// TIA Portal V17 export
// export: Created 2022-07-20T06:59:44.9663361Z, ExportSetting WithDefaults, DisplayName Totally Integrated Automation Portal, DisplayVersion V17, DisplayName TIA Portal Openness, DisplayVersion V17, DisplayName TIA Portal Version Control Interface, DisplayVersion V17, DisplayName SINAMICS Startdrive Advanced, DisplayVersion V17, DisplayName SINAMICS Startdrive G130, G150, S120, S150, SINAMICS MV, S210, DisplayVersion V17, DisplayName SINAMICS Startdrive G110M, G120, G120C, G120D, G120P, G115D, DisplayVersion V17, DisplayName STEP 7 Professional, DisplayVersion V17, DisplayName STEP 7 Safety, DisplayVersion V17, DisplayName WinCC Advanced, DisplayVersion V17
FUNCTION_BLOCK "FB10079_UvDryer"   // FB10079, LAD
{ S7_Optimized_Access := 'TRUE' }
VERSION : 0.1
// stored: AutoNumber false, IsIECCheckEnabled false, IsRetainMemResEnabled false, MemoryReserve 100, SetENOAutomatically false, UDAEnableTagReadback false
   VAR_INPUT
      UvDryer_Disable : Bool;
      Shutter_MotorInError : Bool;
      Shutter_PWMSetPoint : Real;
      Shutter_SensorClosed : Bool;
      Shutter_RequestInitialization : Bool;
      Shutter_RequestOpen : Bool;
      Shutter_RequestClose : Bool;
      Shutter_PWMCardInError : Bool;
      AirExtractor_ScalingShutterOpen : "stAirExtractorScalingParameters";
      AirExtractor_ScalingShutterClosed : "stAirExtractorScalingParameters";
      AirExtractor_PWMMinFrequenceValue : Real;
      AirExtractor_PWMMaxFrequenceValue : Real;
      AirExtractor_RequestActive : Bool;
      UvLamp_ThermalFuse : Bool;
      UvLamp_LampReady : Bool;
      UvLamp_LampWarning : Bool;
      UvLamp_LampError : Bool;
      UvLamp_FeedbackTensionOrErrorCode : Int;
      UvLamp_SetPoint : Real;
      TransportActivated : Bool;
      PowerOnBay : Bool;
   END_VAR
   VAR_OUTPUT
      Shutter_InitializeShutter : Bool;
      Shutter_OpenShutter : Bool;
      Shutter_CloseShutter : Bool;
      Shutter_PWMValue : Real;
      Shutter_ResetPWMCard : Bool;
      Shutter_InError : Bool;
      Shutter_Initialized : Bool;
      Shutter_Opened : Bool;
      Shutter_Closed : Bool;
      AirExtractor_Active : Bool;
      AirExtractor_PWMValue : Real;
      AirExtractor_AnalogValue : Int;
      UvLamp_ActiveLamp : Bool;
      UvLamp_ActivePowerRelay : Bool;
      UvLamp_AnalogValue : Int;
      UvLamp_WarmingUp : Bool;
      UvLamp_ErrorCode : Int;
      UvDryer_Disabled : Bool;
      UvDryer_Ready : Bool;
      UvDryer_Warning : Bool;
      UvDryer_Error : Bool;
      UvDryer_ShutdownInProgress : Bool;
      UvDryer_ShutdownDone : Bool;
      UvDryer_ShutdownTime : Time;
   END_VAR
   VAR_IN_OUT
      UvDryer_RequestStartDryer : Bool;
      UvDryer_RequestShutdown : Bool;
   END_VAR
   VAR
      ShutterMovementManagementStateDiagram : Int;
      DisableShutterStateDiagram : Int;
      AirExtractorManagementStateDiagram : Int;
      R_TRIG_UvDryerDisable : R_TRIG;
      R_TRIG_RequestStartDryer : R_TRIG;
      R_TRIG_ShutterSensorClosed { S7_SetPoint := 'True'} : R_TRIG;
      R_TRIG_RequestInitializeShutter { S7_SetPoint := 'True'} : R_TRIG;
      R_TRIG_RequestOpenShutter { S7_SetPoint := 'True'} : R_TRIG;
      R_TRIG_RequestCloseShutter { S7_SetPoint := 'True'} : R_TRIG;
      R_TRIG_RequestActiveAirExtractor { S7_SetPoint := 'True'} : R_TRIG;
      R_TRIG_RequestShutDown { S7_SetPoint := 'True'} : R_TRIG;
      F_TRIG_RequestStartDryer : F_TRIG;
      F_TRIG_RequestActiveAirExtractor { S7_SetPoint := 'True'} : F_TRIG;
      F_TRIG_PowerOnBay { S7_SetPoint := 'True'} : F_TRIG;
      F_TRIG_TransportActivated { S7_SetPoint := 'True'} : F_TRIG;
      F_TRIG_ShutterSensorClose { S7_SetPoint := 'True'} : F_TRIG;
      F_TRIG_ShutterMotorInError { S7_SetPoint := 'True'} : F_TRIG;
      F_TRIG_UvDryerInError { S7_SetPoint := 'True'} : F_TRIG;
      TON_ShutdownTimer { S7_SetPoint := 'True'} : TON_TIME;
      TON_ShutterMovement { S7_SetPoint := 'True'} : TON_TIME;
      FB10073_LampUVErrorManager_Instance { S7_SetPoint := 'True'} : "FB10073_LampUVErrorManager";
      UvLamp_FeedbackTensionVolts : Real;
      UvLamp_FeedbackTensionPrctg : Real;
   END_VAR
   VAR CONSTANT
      WAIT_FOR_MOVEMENT_REQUEST : Int := 0;
      INITIALIZE_SHUTTER : Int := 10;
      OPEN_SHUTTER : Int := 20;
      CLOSE_SHUTTER : Int := 30;
      MOVEMENT_DONE : Int := 40;
      "==========" : Bool;
      WAIT_FOR_AIR_EXTRACTOR_REQUEST : Int := 0;
      ACTIVE_AIR_EXTRACTOR : Int := 10;
      SHUTDOWN_AIR_EXTRACTOR_IN_PROGRESS : Int := 20;
      ACTIVE_MANUAL_AIR_EXTRACTOR : Int := 30;
      REQUEST_DONE : Int := 40;
   END_VAR
BEGIN

REGION Network 1 (SCL): First Scan
   IF "FirstScan" THEN
       #Shutter_Initialized := FALSE;
       #Shutter_Opened := FALSE;
       #Shutter_Closed := FALSE;
       #ShutterMovementManagementStateDiagram := 0;
   END_IF;
END_REGION

REGION Network 2 (SCL): Edge Signals & Timers
   REGION EDGE SIGNALS
       #R_TRIG_UvDryerDisable(CLK := #UvDryer_Disable);
       #R_TRIG_RequestStartDryer(CLK := #UvDryer_RequestStartDryer AND NOT(#UvDryer_ShutdownInProgress));
       #R_TRIG_RequestInitializeShutter(CLK := #Shutter_RequestInitialization);
       #R_TRIG_RequestOpenShutter(CLK := #Shutter_RequestOpen);
       #R_TRIG_RequestCloseShutter(CLK := #Shutter_RequestClose);
       #R_TRIG_ShutterSensorClosed(CLK := #Shutter_SensorClosed);
       #R_TRIG_RequestShutDown(CLK := #UvDryer_RequestShutdown);
       #R_TRIG_RequestActiveAirExtractor(CLK := #AirExtractor_RequestActive);

       #F_TRIG_RequestStartDryer(CLK := #UvDryer_RequestStartDryer);
       #F_TRIG_RequestActiveAirExtractor(CLK := #AirExtractor_RequestActive);
       #F_TRIG_PowerOnBay(CLK := #PowerOnBay);
       #F_TRIG_TransportActivated(CLK := #TransportActivated);
       #F_TRIG_ShutterSensorClose(CLK := #Shutter_SensorClosed);
       #F_TRIG_UvDryerInError(CLK := #UvDryer_Error);
       #F_TRIG_ShutterMotorInError(CLK := #Shutter_InError);
   END_REGION

   REGION TIMERS
       #TON_ShutdownTimer(IN := #UvDryer_ShutdownInProgress AND #PowerOnBay,
                          PT := T#5m,
                          ET => #UvDryer_ShutdownTime);
       #TON_ShutterMovement(IN := (#ShutterMovementManagementStateDiagram = #INITIALIZE_SHUTTER) OR
                            (#ShutterMovementManagementStateDiagram = #OPEN_SHUTTER) OR
                            (#ShutterMovementManagementStateDiagram = #CLOSE_SHUTTER),
                            PT := T#10s);
   END_REGION
END_REGION

REGION Network 3 (SCL): Uv Dryer Commands Management
   IF #F_TRIG_PowerOnBay.Q OR #F_TRIG_UvDryerInError.Q OR #F_TRIG_ShutterMotorInError.Q OR #UvDryer_Disable OR #UvDryer_ShutdownInProgress THEN
       #UvDryer_RequestStartDryer := FALSE;
   END_IF;
END_REGION

REGION Network 4 (SCL): Shutter Management
   CASE #ShutterMovementManagementStateDiagram OF
       #WAIT_FOR_MOVEMENT_REQUEST:
           IF (#R_TRIG_RequestStartDryer.Q OR #R_TRIG_RequestInitializeShutter.Q) AND NOT (#UvDryer_Disable) THEN
               #ShutterMovementManagementStateDiagram := #INITIALIZE_SHUTTER;
           ELSIF #R_TRIG_RequestOpenShutter.Q AND #Shutter_SensorClosed AND #TransportActivated AND #Shutter_Initialized THEN
               #Shutter_Opened := FALSE;
               #Shutter_Closed := FALSE;
               #ShutterMovementManagementStateDiagram := #OPEN_SHUTTER;
           ELSIF (#R_TRIG_RequestCloseShutter.Q OR #F_TRIG_TransportActivated.Q OR (#R_TRIG_UvDryerDisable.Q AND #Shutter_InError)) AND NOT (#Shutter_SensorClosed) THEN
               #Shutter_Opened := FALSE;
               #Shutter_Closed := FALSE;
               #ShutterMovementManagementStateDiagram := #CLOSE_SHUTTER;
           END_IF;
       #INITIALIZE_SHUTTER:
           #Shutter_InitializeShutter := TRUE;
           #Shutter_PWMValue := #Shutter_PWMSetPoint;
           IF #R_TRIG_ShutterSensorClosed.Q THEN
               RESET_TIMER(#TON_ShutterMovement);
               #Shutter_InitializeShutter := FALSE;
               #Shutter_Initialized := TRUE;
               #Shutter_Opened := FALSE;
               #Shutter_Closed := TRUE;
               #ShutterMovementManagementStateDiagram := #MOVEMENT_DONE;
           END_IF;
       #OPEN_SHUTTER:
           #Shutter_OpenShutter := TRUE;
           #Shutter_PWMValue := #Shutter_PWMSetPoint;
           IF #F_TRIG_ShutterSensorClose.Q THEN
               RESET_TIMER(#TON_ShutterMovement);
               #Shutter_OpenShutter := FALSE;
               #Shutter_Opened := TRUE;
               #Shutter_Closed := FALSE;
               #ShutterMovementManagementStateDiagram := #MOVEMENT_DONE;
           END_IF;
       #CLOSE_SHUTTER:
           #Shutter_CloseShutter := TRUE;
           #Shutter_PWMValue := #Shutter_PWMSetPoint;
           IF #R_TRIG_ShutterSensorClosed.Q THEN
               RESET_TIMER(#TON_ShutterMovement);
               #Shutter_CloseShutter := FALSE;
               #Shutter_Opened := FALSE;
               #Shutter_Closed := TRUE;
               #ShutterMovementManagementStateDiagram := #MOVEMENT_DONE;
           END_IF;
       #MOVEMENT_DONE:
           #ShutterMovementManagementStateDiagram := #WAIT_FOR_MOVEMENT_REQUEST;
   END_CASE;
END_REGION

REGION Network 5 (SCL): Air Extractor Management
   IF #R_TRIG_RequestStartDryer.Q AND NOT (#UvDryer_Disable) THEN
       #UvDryer_ShutdownDone := FALSE;
       #AirExtractorManagementStateDiagram := #ACTIVE_AIR_EXTRACTOR;
   ELSIF
       (#R_TRIG_RequestShutDown.Q AND NOT (#UvDryer_Disabled)) OR
       (#F_TRIG_RequestStartDryer.Q AND NOT (#UvDryer_Disabled)) OR
       (#R_TRIG_UvDryerDisable.Q AND (#AirExtractorManagementStateDiagram = #ACTIVE_AIR_EXTRACTOR OR #AirExtractorManagementStateDiagram = #ACTIVE_MANUAL_AIR_EXTRACTOR))
   THEN
       #AirExtractorManagementStateDiagram := #SHUTDOWN_AIR_EXTRACTOR_IN_PROGRESS;
   END_IF;

   CASE #AirExtractorManagementStateDiagram OF
       #WAIT_FOR_AIR_EXTRACTOR_REQUEST:
           #UvDryer_ShutdownInProgress := FALSE;
           #AirExtractor_Active := FALSE;
           #AirExtractor_PWMValue := 0;
           #AirExtractor_AnalogValue := 0;

           IF #R_TRIG_RequestActiveAirExtractor.Q AND NOT(#UvDryer_Disable) THEN
               #UvDryer_ShutdownDone := FALSE;
               #AirExtractorManagementStateDiagram := #ACTIVE_MANUAL_AIR_EXTRACTOR;
           END_IF;
       #ACTIVE_AIR_EXTRACTOR:
           #AirExtractor_Active := TRUE;
           IF #Shutter_Closed THEN
               "FC10072_ScalingAirExtraction_VolatgeFeedback"(VoltageFeedback := #UvLamp_FeedbackTensionVolts,
                                                              X_UVPower_Min := #AirExtractor_ScalingShutterClosed.PowerXMin,
                                                              X_UVPower_Max := #AirExtractor_ScalingShutterClosed.PowerXMax,
                                                              Y_AirPower_Min := #AirExtractor_ScalingShutterClosed.PowerAirYMin,
                                                              Y_AirPower_Max := #AirExtractor_ScalingShutterClosed.PowerAirYMax,
                                                              PWM_Minimum := #AirExtractor_PWMMinFrequenceValue,
                                                              PWM_Maximum := #AirExtractor_PWMMaxFrequenceValue,
                                                              Analogical_Value => #AirExtractor_AnalogValue,
                                                              PWM_FrequenceValue => #AirExtractor_PWMValue);
           ELSIF #Shutter_Opened THEN
               "FC10072_ScalingAirExtraction_VolatgeFeedback"(VoltageFeedback := #UvLamp_FeedbackTensionVolts,
                                                              X_UVPower_Min := #AirExtractor_ScalingShutterOpen.PowerXMin,
                                                              X_UVPower_Max := #AirExtractor_ScalingShutterOpen.PowerXMax,
                                                              Y_AirPower_Min := #AirExtractor_ScalingShutterOpen.PowerAirYMin,
                                                              Y_AirPower_Max := #AirExtractor_ScalingShutterOpen.PowerAirYMax,
                                                              PWM_Minimum := #AirExtractor_PWMMinFrequenceValue,
                                                              PWM_Maximum := #AirExtractor_PWMMaxFrequenceValue,
                                                              Analogical_Value => #AirExtractor_AnalogValue,
                                                              PWM_FrequenceValue => #AirExtractor_PWMValue);
           END_IF;


           IF #R_TRIG_RequestShutDown.Q OR #F_TRIG_RequestStartDryer.Q THEN
               #AirExtractorManagementStateDiagram := #SHUTDOWN_AIR_EXTRACTOR_IN_PROGRESS;
           END_IF;
       #SHUTDOWN_AIR_EXTRACTOR_IN_PROGRESS:
           #AirExtractor_Active := TRUE;

           "FC10072_ScalingAirExtraction_VolatgeFeedback"(VoltageFeedback := #AirExtractor_ScalingShutterClosed.PowerXMax,
                                                          X_UVPower_Min := #AirExtractor_ScalingShutterClosed.PowerXMin,
                                                          X_UVPower_Max := #AirExtractor_ScalingShutterClosed.PowerXMax,
                                                          Y_AirPower_Min := #AirExtractor_ScalingShutterClosed.PowerAirYMin,
                                                          Y_AirPower_Max := #AirExtractor_ScalingShutterClosed.PowerAirYMax,
                                                          PWM_Minimum := #AirExtractor_PWMMinFrequenceValue,
                                                          PWM_Maximum := #AirExtractor_PWMMaxFrequenceValue,
                                                          Analogical_Value => #AirExtractor_AnalogValue,
                                                          PWM_FrequenceValue => #AirExtractor_PWMValue);
           IF #TON_ShutdownTimer.Q THEN
               #AirExtractor_Active := FALSE;
               #UvDryer_ShutdownDone := TRUE;
               #AirExtractorManagementStateDiagram := #REQUEST_DONE;
           END_IF;
       #ACTIVE_MANUAL_AIR_EXTRACTOR:
           #AirExtractor_Active := TRUE;
           "FC10072_ScalingAirExtraction_VolatgeFeedback"(VoltageFeedback := #AirExtractor_ScalingShutterClosed.PowerXMin,
                                                          X_UVPower_Min := #AirExtractor_ScalingShutterClosed.PowerXMin,
                                                          X_UVPower_Max := #AirExtractor_ScalingShutterClosed.PowerXMax,
                                                          Y_AirPower_Min := #AirExtractor_ScalingShutterClosed.PowerAirYMin,
                                                          Y_AirPower_Max := #AirExtractor_ScalingShutterClosed.PowerAirYMax,
                                                          PWM_Minimum := #AirExtractor_PWMMinFrequenceValue,
                                                          PWM_Maximum := #AirExtractor_PWMMaxFrequenceValue,
                                                          Analogical_Value => #AirExtractor_AnalogValue,
                                                          PWM_FrequenceValue => #AirExtractor_PWMValue);
           IF #F_TRIG_RequestActiveAirExtractor.Q THEN
               #AirExtractorManagementStateDiagram := #REQUEST_DONE;
           END_IF;
       #REQUEST_DONE:
           #AirExtractor_Active := FALSE;
           #AirExtractor_PWMValue := 0;
           #AirExtractor_AnalogValue := 0;
           #AirExtractorManagementStateDiagram := #WAIT_FOR_AIR_EXTRACTOR_REQUEST;
   END_CASE;
END_REGION

REGION Network 6 (SCL): Uv Lamp Management
   IF NOT(#UvDryer_Disable) THEN //Uv Lamp Requests And SetPoint Management
       IF #UvDryer_RequestStartDryer AND #Shutter_Initialized AND #AirExtractor_Active THEN
           #UvLamp_ActiveLamp := TRUE;
           IF #Shutter_Opened THEN
               "FC10010_ScalingPercentageToAnalog"(SetPoint := #UvLamp_SetPoint,
                                                   AnalogValue => #UvLamp_AnalogValue);
           ELSIF #Shutter_Closed THEN
               #UvLamp_AnalogValue := 0;
           ELSE
               #UvLamp_AnalogValue := 0;
           END_IF;
       ELSE
           #UvLamp_ActiveLamp := FALSE;
           #UvLamp_AnalogValue := 0;
       END_IF;

       //Emergency Stop Management
       IF #PowerOnBay THEN
           #UvLamp_ActivePowerRelay := TRUE;
       ELSE
           #UvLamp_ActivePowerRelay := FALSE;
       END_IF;
   ELSE
       #UvLamp_ActivePowerRelay := FALSE;
       #UvLamp_ActiveLamp := FALSE;
       #UvLamp_AnalogValue := 0;
   END_IF;
END_REGION

REGION Network 7 (SCL): Uv Dryer States Management
   REGION UV LAMP STATES
       #FB10073_LampUVErrorManager_Instance(ReadySignal := #UvLamp_LampReady,
                                            WarningSignal := #UvLamp_LampWarning,
                                            ErrorSignal := #UvLamp_LampError,
                                            ErrorCodeAnalog := #UvLamp_FeedbackTensionOrErrorCode,
                                            ErrorCode => #UvLamp_ErrorCode);
       #UvLamp_FeedbackTensionPrctg := INT_TO_REAL(#UvLamp_FeedbackTensionOrErrorCode) / 276.48;
       #UvLamp_FeedbackTensionVolts := #UvLamp_FeedbackTensionPrctg * 10.0;
       #UvLamp_WarmingUp := NOT (#UvLamp_LampReady) AND #UvLamp_LampError AND #UvDryer_RequestStartDryer;
   END_REGION

   REGION SHUTTER
       IF #TON_ShutterMovement.Q OR NOT(#Shutter_MotorInError) THEN
           #Shutter_InitializeShutter := FALSE;
           #Shutter_OpenShutter := FALSE;
           #Shutter_CloseShutter := FALSE;
           #ShutterMovementManagementStateDiagram := #WAIT_FOR_MOVEMENT_REQUEST;
           #Shutter_InError := TRUE;
       END_IF;

       IF #Shutter_PWMCardInError THEN
           #Shutter_ResetPWMCard := "Clock_0.5Hz";
       ELSE
           #Shutter_ResetPWMCard := FALSE;
       END_IF;

       IF #F_TRIG_RequestStartDryer.Q OR #R_TRIG_UvDryerDisable.Q THEN
           #Shutter_Initialized := FALSE;
       END_IF;
   END_REGION 

   REGION UV DRYER
       #UvDryer_Ready := #UvLamp_LampReady;

       #UvDryer_Warning := NOT (#UvLamp_LampWarning); //To Change When It Will Be Really Wired

       #UvDryer_Error := #UvLamp_LampError;

       #UvDryer_Disabled := #UvDryer_Disable AND
       (NOT (#UvLamp_ActivePowerRelay) AND NOT (#UvLamp_ActiveLamp) AND #UvLamp_AnalogValue = 0) AND
       (NOT (#AirExtractor_Active) AND #AirExtractor_PWMValue = 0 AND #AirExtractor_AnalogValue = 0);

       #UvDryer_ShutdownInProgress := #AirExtractorManagementStateDiagram = #SHUTDOWN_AIR_EXTRACTOR_IN_PROGRESS;

       IF #TON_ShutdownTimer.Q THEN
           #UvDryer_ShutdownDone := TRUE;
       ELSIF #TON_ShutdownTimer.ET > T#0s THEN
           #UvDryer_ShutdownDone := FALSE;
       END_IF;
   END_REGION
END_REGION
END_FUNCTION_BLOCK
